// SIMATIC S7-200 project (STEP 7-Micro/WIN), CPU 224 REL 02.01

ORGANIZATION_BLOCK MAIN:OB1
TITLE=PROGRAM COMMENTS
BEGIN
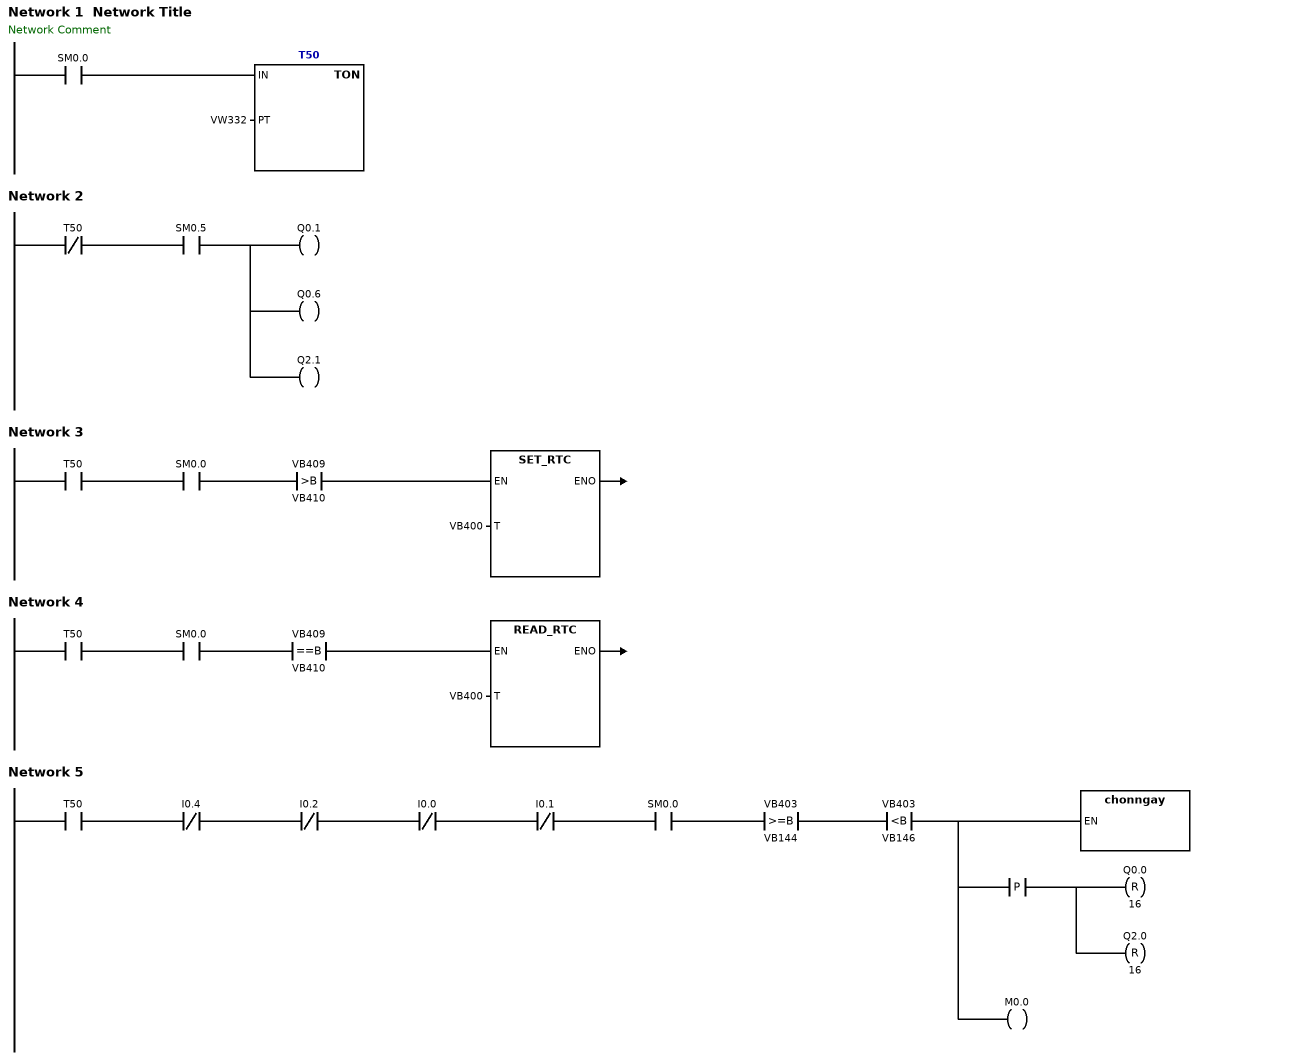
Network 1 // Network Title
// Network Comment
LD     SM0.0
TON    T50, VW332
Network 2
LDN    T50
A      SM0.5
=      Q0.1
=      Q0.6
=      Q2.1
Network 3
LD     T50
A      SM0.0
AB>    VB409, VB410
TODW   VB400
Network 4
LD     T50
A      SM0.0
AB=    VB409, VB410
TODR   VB400
Network 5
LD     T50
AN     I0.4
AN     I0.2
AN     I0.0
AN     I0.1
A      SM0.0
AB>=   VB403, VB144
AB<    VB403, VB146
LPS
CALL   chonngay:SBR11
EU
R      Q0.0, 16
R      Q2.0, 16
LPP
=      M0.0
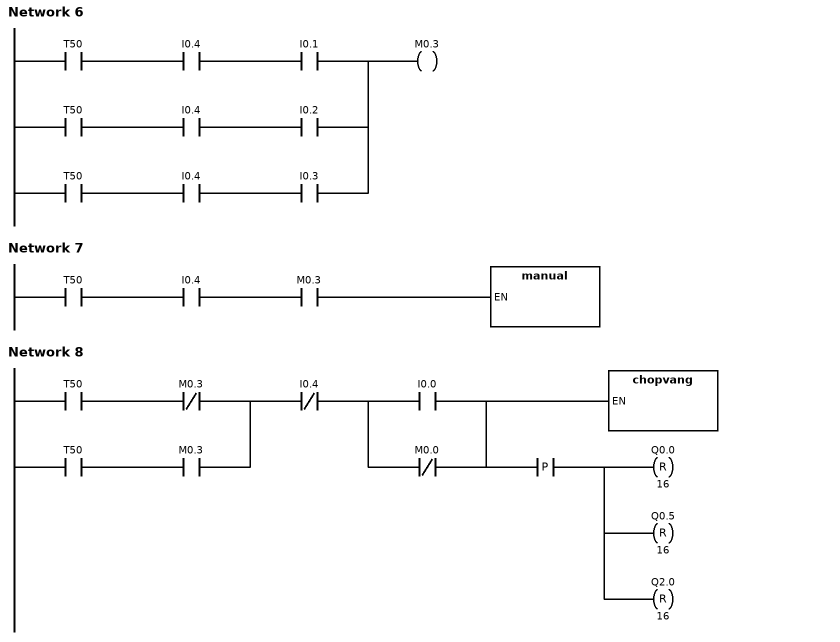
Network 6
LD     T50
A      I0.4
A      I0.1
LD     T50
A      I0.4
A      I0.2
OLD
LD     T50
A      I0.4
A      I0.3
OLD
=      M0.3
Network 7
LD     T50
A      I0.4
A      M0.3
CALL   manual:SBR2
Network 8
LD     T50
AN     M0.3
LD     T50
A      M0.3
OLD
AN     I0.4
LD     I0.0
ON     M0.0
ALD
CALL   chopvang:SBR1
EU
R      Q0.0, 16
R      Q0.5, 16
R      Q2.0, 16
END_ORGANIZATION_BLOCK

SUBROUTINE_BLOCK tudong2phase:SBR0
TITLE=SUBROUTINE COMMENTS
BEGIN
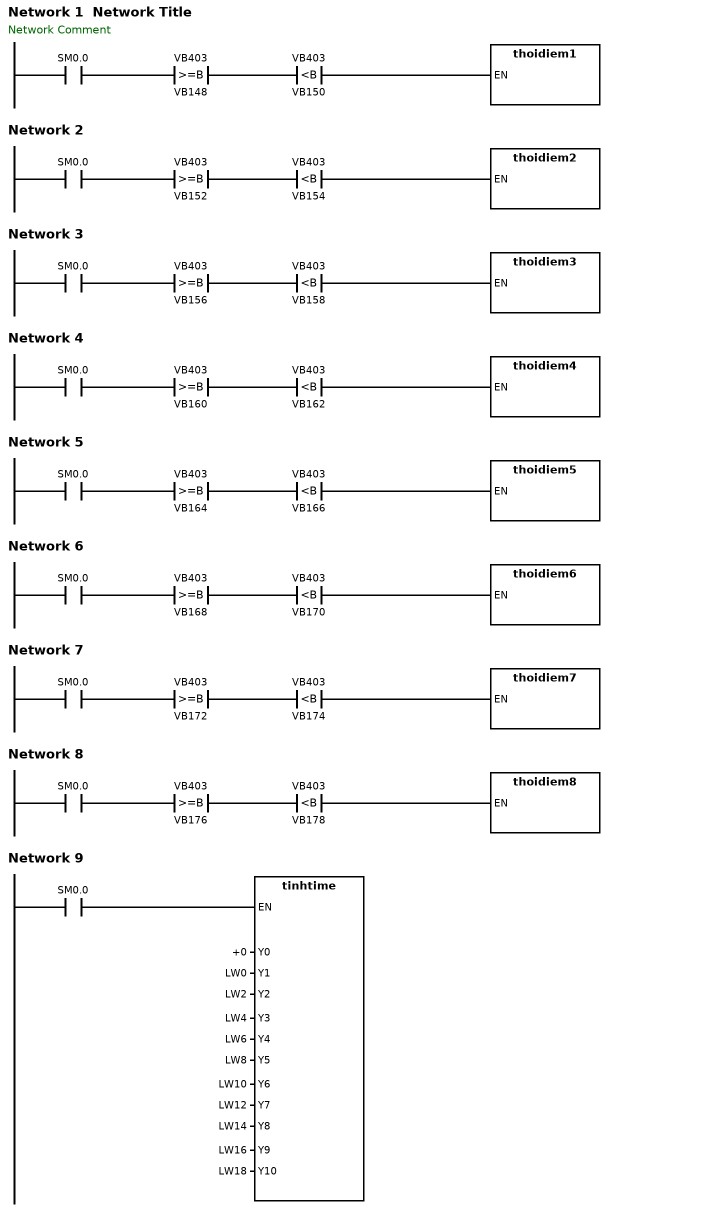
Network 1 // Network Title
// Network Comment
LD     SM0.0
AB>=   VB403, VB148
AB<    VB403, VB150
CALL   thoidiem1:SBR3
Network 2
LD     SM0.0
AB>=   VB403, VB152
AB<    VB403, VB154
CALL   thoidiem2:SBR4
Network 3
LD     SM0.0
AB>=   VB403, VB156
AB<    VB403, VB158
CALL   thoidiem3:SBR5
Network 4
LD     SM0.0
AB>=   VB403, VB160
AB<    VB403, VB162
CALL   thoidiem4:SBR6
Network 5
LD     SM0.0
AB>=   VB403, VB164
AB<    VB403, VB166
CALL   thoidiem5:SBR7
Network 6
LD     SM0.0
AB>=   VB403, VB168
AB<    VB403, VB170
CALL   thoidiem6:SBR8
Network 7
LD     SM0.0
AB>=   VB403, VB172
AB<    VB403, VB174
CALL   thoidiem7:SBR9
Network 8
LD     SM0.0
AB>=   VB403, VB176
AB<    VB403, VB178
CALL   thoidiem8:SBR14
Network 9
LD     SM0.0
CALL   tinhtime:SBR16, +0, LW0, LW2, LW4, LW6, LW8, LW10, LW12, LW14, LW16, LW18
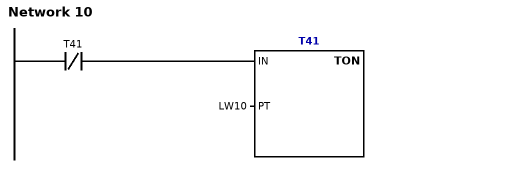
Network 10
LDN    T41
TON    T41, LW10
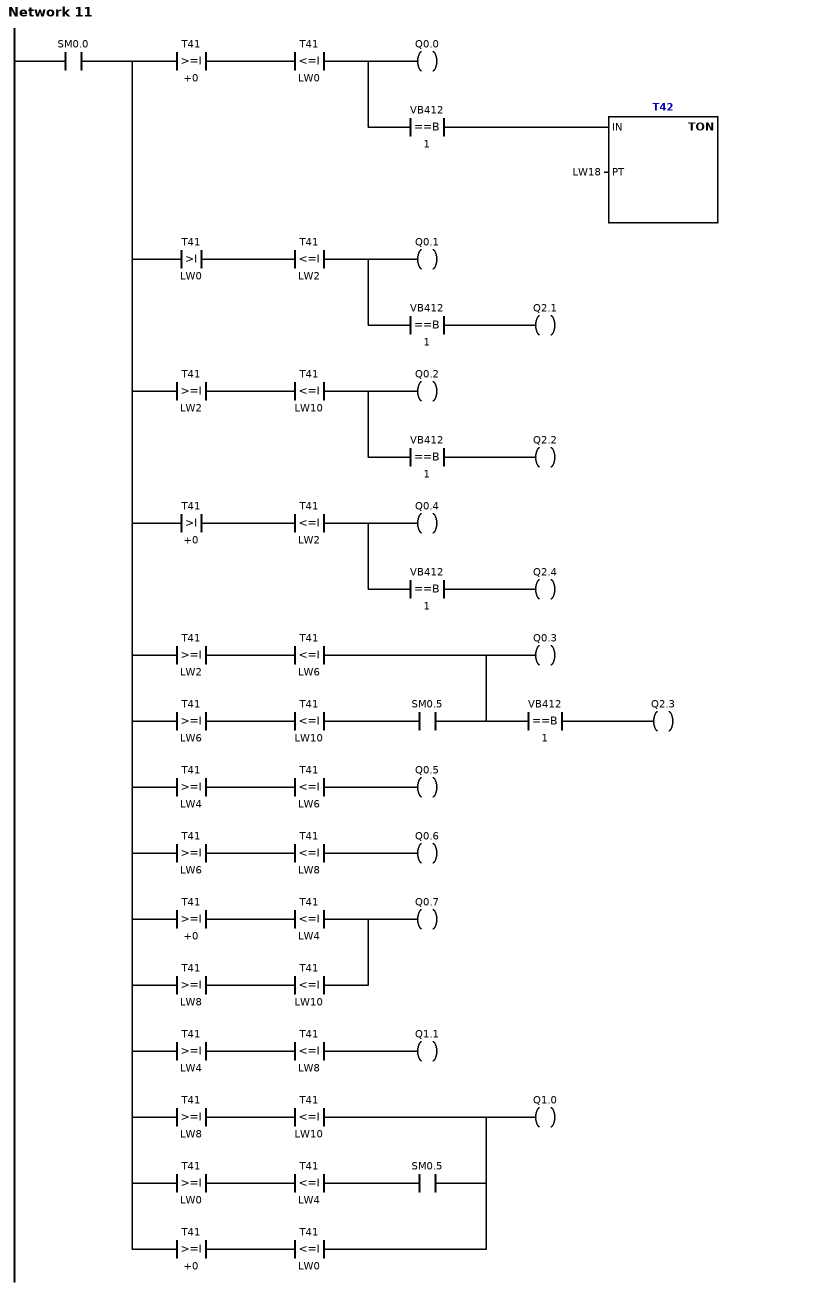
Network 11
LD     SM0.0
LPS
AW>=   T41, +0
AW<=   T41, LW0
=      Q0.0
AB=    VB412, 1
TON    T42, LW18
LRD
AW>    T41, LW0
AW<=   T41, LW2
=      Q0.1
AB=    VB412, 1
=      Q2.1
LRD
AW>=   T41, LW2
AW<=   T41, LW10
=      Q0.2
AB=    VB412, 1
=      Q2.2
LRD
AW>    T41, +0
AW<=   T41, LW2
=      Q0.4
AB=    VB412, 1
=      Q2.4
LRD
LDW>=  T41, LW2
AW<=   T41, LW6
LDW>=  T41, LW6
AW<=   T41, LW10
A      SM0.5
OLD
ALD
=      Q0.3
AB=    VB412, 1
=      Q2.3
LRD
LPS
AW>=   T41, LW4
AW<=   T41, LW6
=      Q0.5
LPP
AW>=   T41, LW6
AW<=   T41, LW8
=      Q0.6
LRD
LDW>=  T41, +0
AW<=   T41, LW4
LDW>=  T41, LW8
AW<=   T41, LW10
OLD
ALD
=      Q0.7
LRD
AW>=   T41, LW4
AW<=   T41, LW8
=      Q1.1
LPP
LDW>=  T41, LW8
AW<=   T41, LW10
LDW>=  T41, LW0
AW<=   T41, LW4
A      SM0.5
OLD
LDW>=  T41, +0
AW<=   T41, LW0
OLD
ALD
=      Q1.0
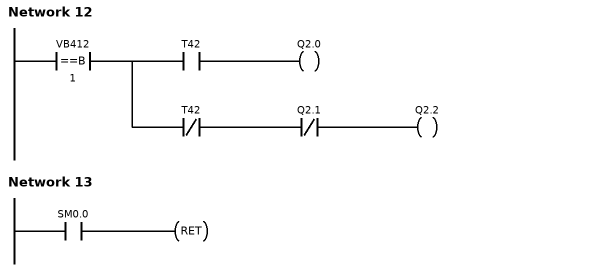
Network 12
LDB=   VB412, 1
LPS
A      T42
=      Q2.0
LPP
AN     T42
AN     Q2.1
=      Q2.2
Network 13
LD     SM0.0
CRET
END_SUBROUTINE_BLOCK

SUBROUTINE_BLOCK chopvang:SBR1
TITLE=
BEGIN
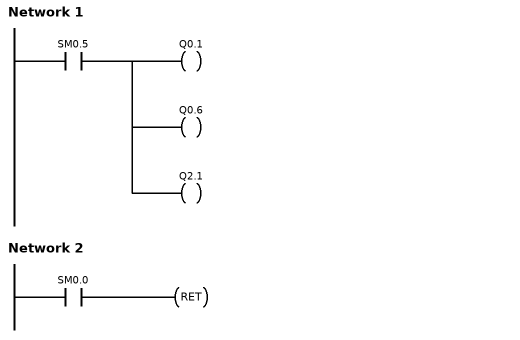
Network 1
LD     SM0.5
=      Q0.1
=      Q0.6
=      Q2.1
Network 2
LD     SM0.0
CRET
END_SUBROUTINE_BLOCK

SUBROUTINE_BLOCK manual:SBR2
TITLE=
BEGIN
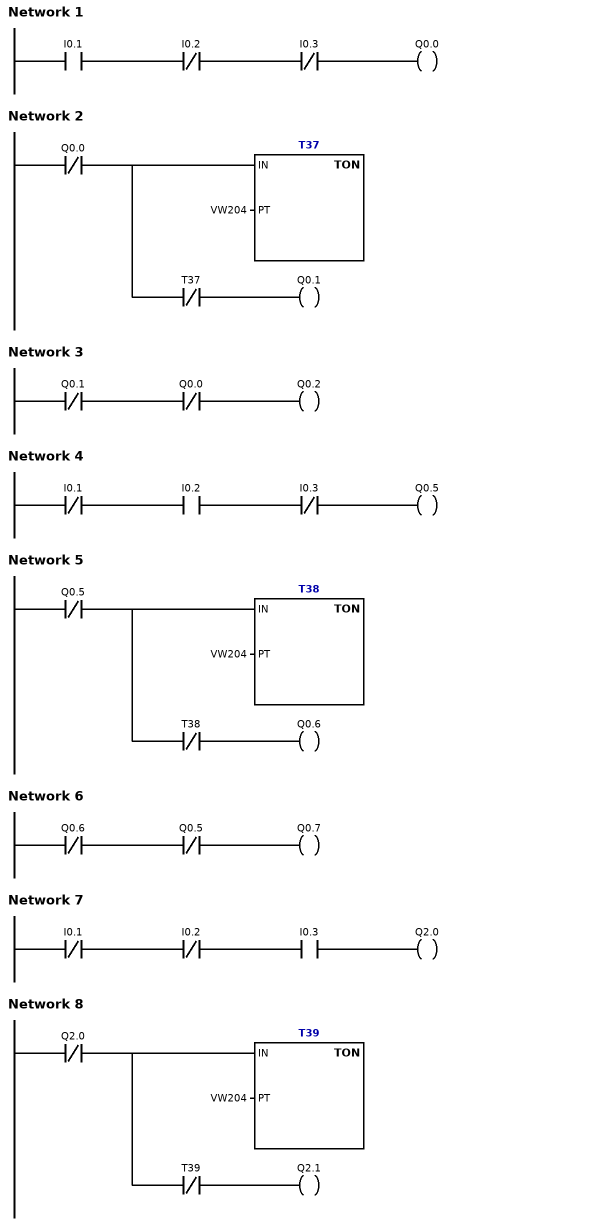
Network 1
LD     I0.1
AN     I0.2
AN     I0.3
=      Q0.0
Network 2
LDN    Q0.0
TON    T37, VW204
AN     T37
=      Q0.1
Network 3
LDN    Q0.1
AN     Q0.0
=      Q0.2
Network 4
LDN    I0.1
A      I0.2
AN     I0.3
=      Q0.5
Network 5
LDN    Q0.5
TON    T38, VW204
AN     T38
=      Q0.6
Network 6
LDN    Q0.6
AN     Q0.5
=      Q0.7
Network 7
LDN    I0.1
AN     I0.2
A      I0.3
=      Q2.0
Network 8
LDN    Q2.0
TON    T39, VW204
AN     T39
=      Q2.1
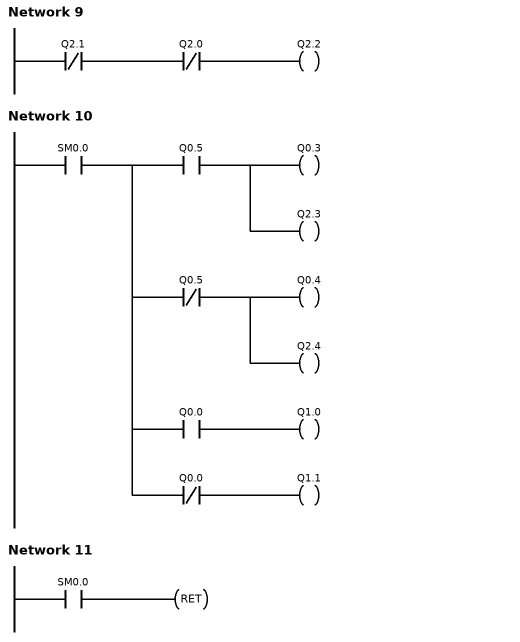
Network 9
LDN    Q2.1
AN     Q2.0
=      Q2.2
Network 10
LD     SM0.0
LPS
A      Q0.5
=      Q0.3
=      Q2.3
LRD
AN     Q0.5
=      Q0.4
=      Q2.4
LPP
LPS
A      Q0.0
=      Q1.0
LPP
AN     Q0.0
=      Q1.1
Network 11
LD     SM0.0
CRET
END_SUBROUTINE_BLOCK

SUBROUTINE_BLOCK thoidiem1:SBR3
TITLE=
BEGIN
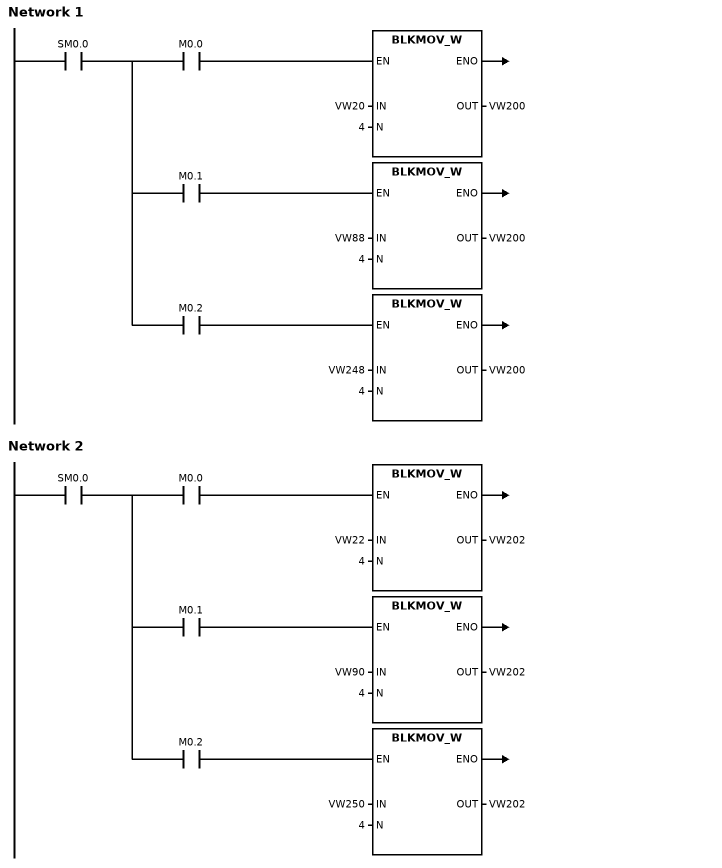
Network 1
LD     SM0.0
LPS
A      M0.0
BMW    VW20, VW200, 4
LRD
A      M0.1
BMW    VW88, VW200, 4
LPP
A      M0.2
BMW    VW248, VW200, 4
Network 2
LD     SM0.0
LPS
A      M0.0
BMW    VW22, VW202, 4
LRD
A      M0.1
BMW    VW90, VW202, 4
LPP
A      M0.2
BMW    VW250, VW202, 4
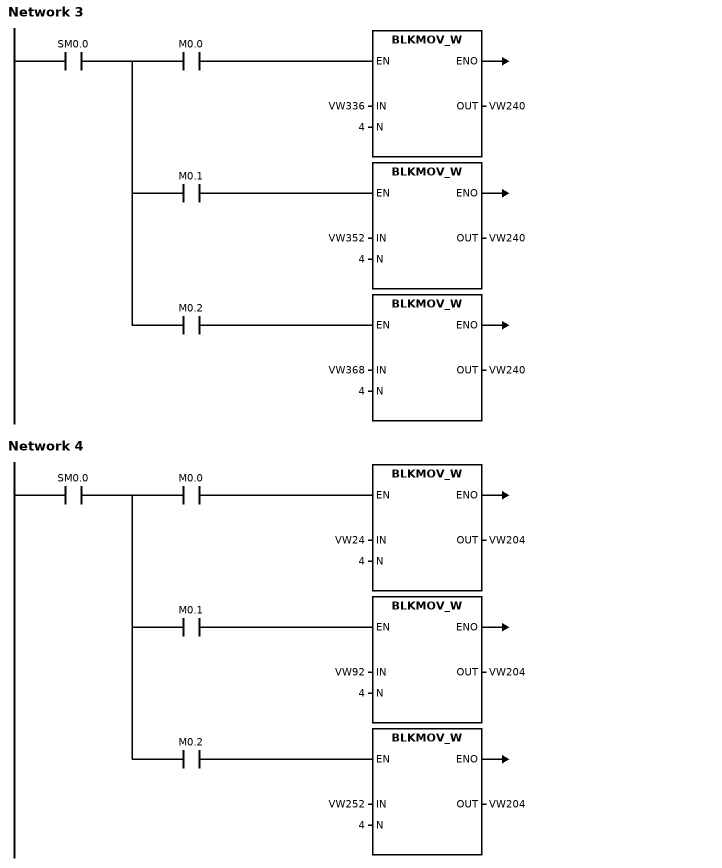
Network 3
LD     SM0.0
LPS
A      M0.0
BMW    VW336, VW240, 4
LRD
A      M0.1
BMW    VW352, VW240, 4
LPP
A      M0.2
BMW    VW368, VW240, 4
Network 4
LD     SM0.0
LPS
A      M0.0
BMW    VW24, VW204, 4
LRD
A      M0.1
BMW    VW92, VW204, 4
LPP
A      M0.2
BMW    VW252, VW204, 4
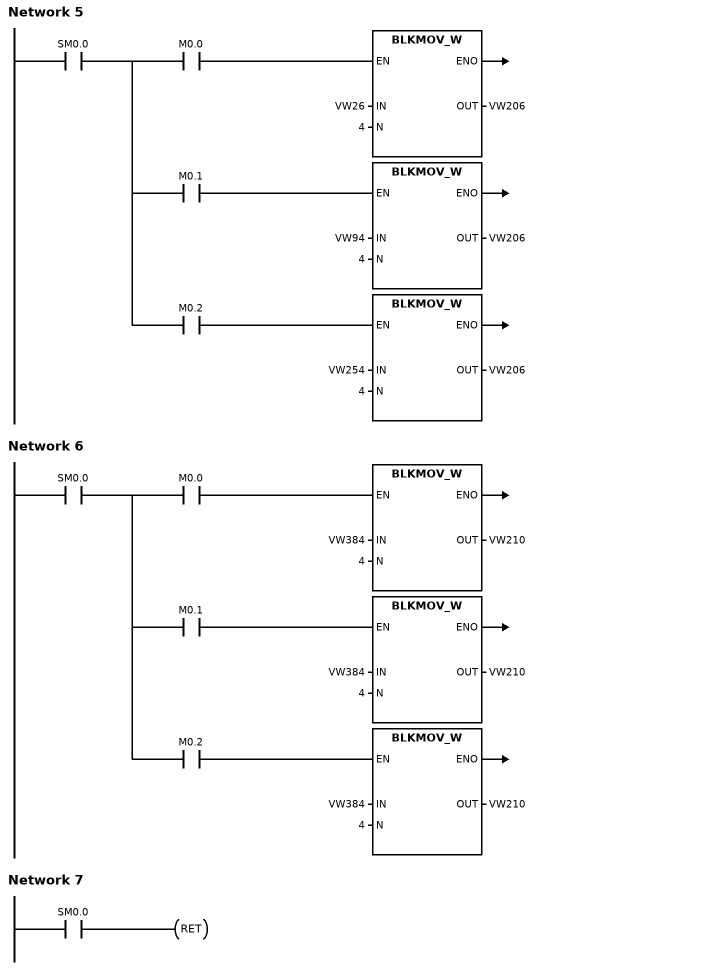
Network 5
LD     SM0.0
LPS
A      M0.0
BMW    VW26, VW206, 4
LRD
A      M0.1
BMW    VW94, VW206, 4
LPP
A      M0.2
BMW    VW254, VW206, 4
Network 6
LD     SM0.0
LPS
A      M0.0
BMW    VW384, VW210, 4
LRD
A      M0.1
BMW    VW384, VW210, 4
LPP
A      M0.2
BMW    VW384, VW210, 4
Network 7
LD     SM0.0
CRET
END_SUBROUTINE_BLOCK

SUBROUTINE_BLOCK thoidiem2:SBR4
TITLE=
BEGIN
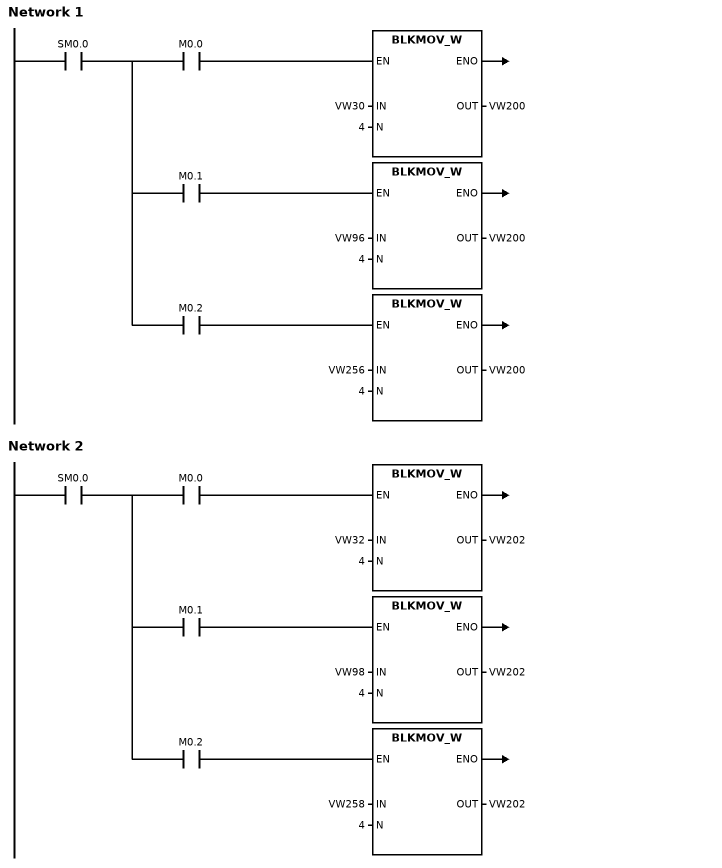
Network 1
LD     SM0.0
LPS
A      M0.0
BMW    VW30, VW200, 4
LRD
A      M0.1
BMW    VW96, VW200, 4
LPP
A      M0.2
BMW    VW256, VW200, 4
Network 2
LD     SM0.0
LPS
A      M0.0
BMW    VW32, VW202, 4
LRD
A      M0.1
BMW    VW98, VW202, 4
LPP
A      M0.2
BMW    VW258, VW202, 4
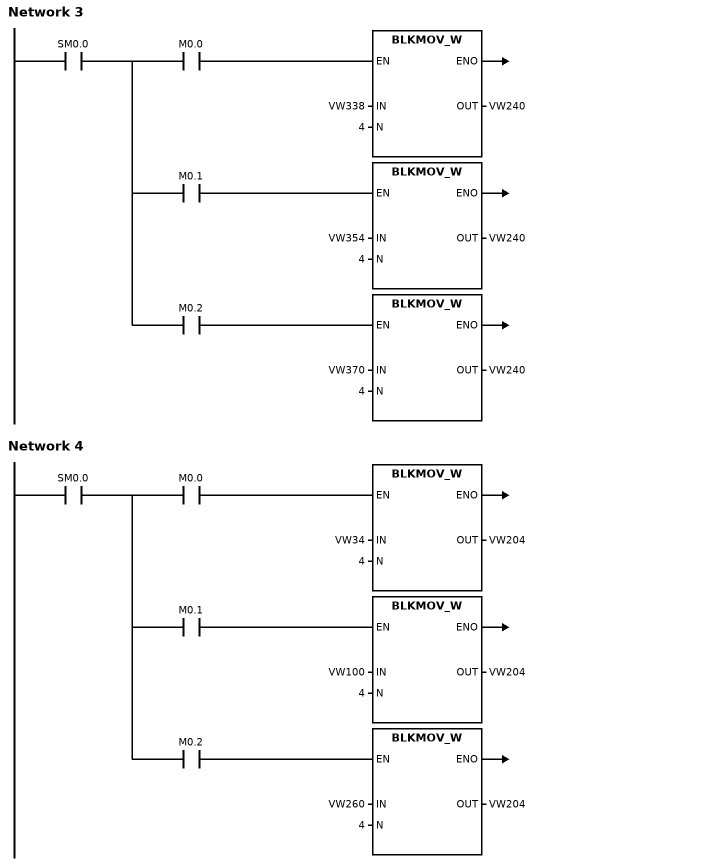
Network 3
LD     SM0.0
LPS
A      M0.0
BMW    VW338, VW240, 4
LRD
A      M0.1
BMW    VW354, VW240, 4
LPP
A      M0.2
BMW    VW370, VW240, 4
Network 4
LD     SM0.0
LPS
A      M0.0
BMW    VW34, VW204, 4
LRD
A      M0.1
BMW    VW100, VW204, 4
LPP
A      M0.2
BMW    VW260, VW204, 4
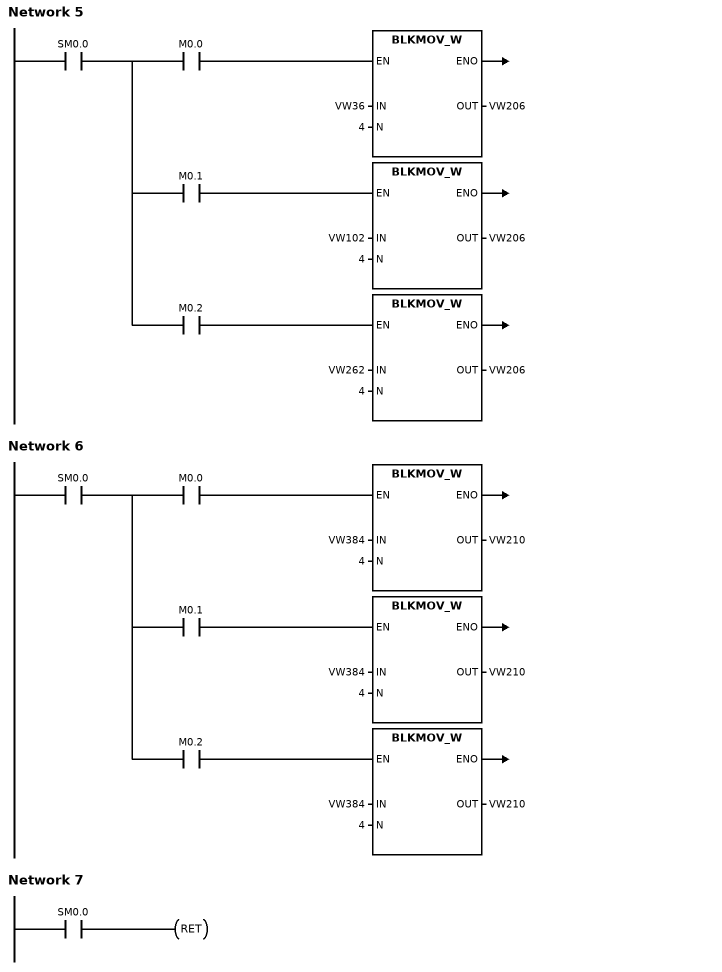
Network 5
LD     SM0.0
LPS
A      M0.0
BMW    VW36, VW206, 4
LRD
A      M0.1
BMW    VW102, VW206, 4
LPP
A      M0.2
BMW    VW262, VW206, 4
Network 6
LD     SM0.0
LPS
A      M0.0
BMW    VW384, VW210, 4
LRD
A      M0.1
BMW    VW384, VW210, 4
LPP
A      M0.2
BMW    VW384, VW210, 4
Network 7
LD     SM0.0
CRET
END_SUBROUTINE_BLOCK

SUBROUTINE_BLOCK thoidiem3:SBR5
TITLE=
BEGIN
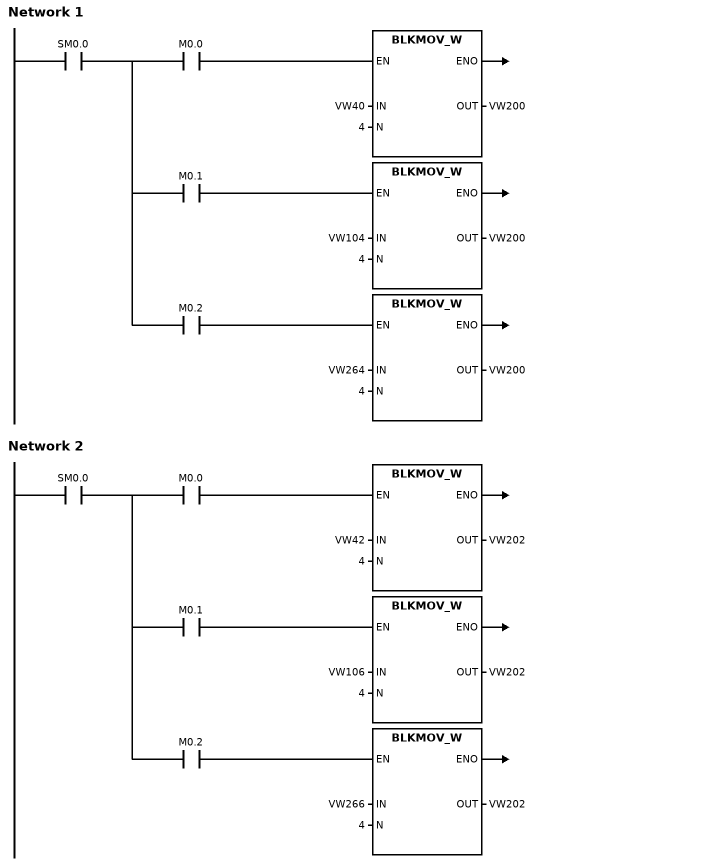
Network 1
LD     SM0.0
LPS
A      M0.0
BMW    VW40, VW200, 4
LRD
A      M0.1
BMW    VW104, VW200, 4
LPP
A      M0.2
BMW    VW264, VW200, 4
Network 2
LD     SM0.0
LPS
A      M0.0
BMW    VW42, VW202, 4
LRD
A      M0.1
BMW    VW106, VW202, 4
LPP
A      M0.2
BMW    VW266, VW202, 4
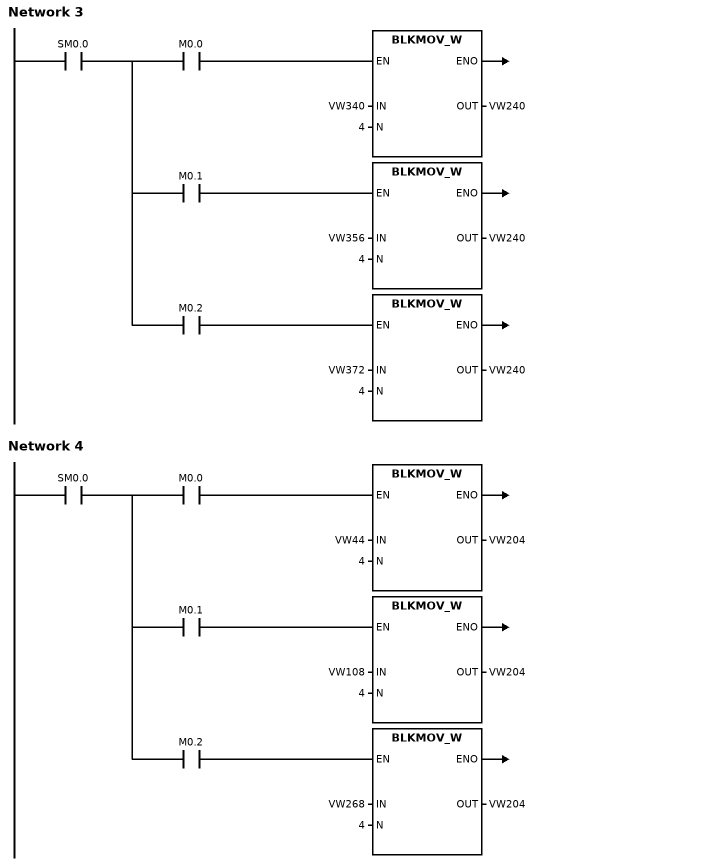
Network 3
LD     SM0.0
LPS
A      M0.0
BMW    VW340, VW240, 4
LRD
A      M0.1
BMW    VW356, VW240, 4
LPP
A      M0.2
BMW    VW372, VW240, 4
Network 4
LD     SM0.0
LPS
A      M0.0
BMW    VW44, VW204, 4
LRD
A      M0.1
BMW    VW108, VW204, 4
LPP
A      M0.2
BMW    VW268, VW204, 4
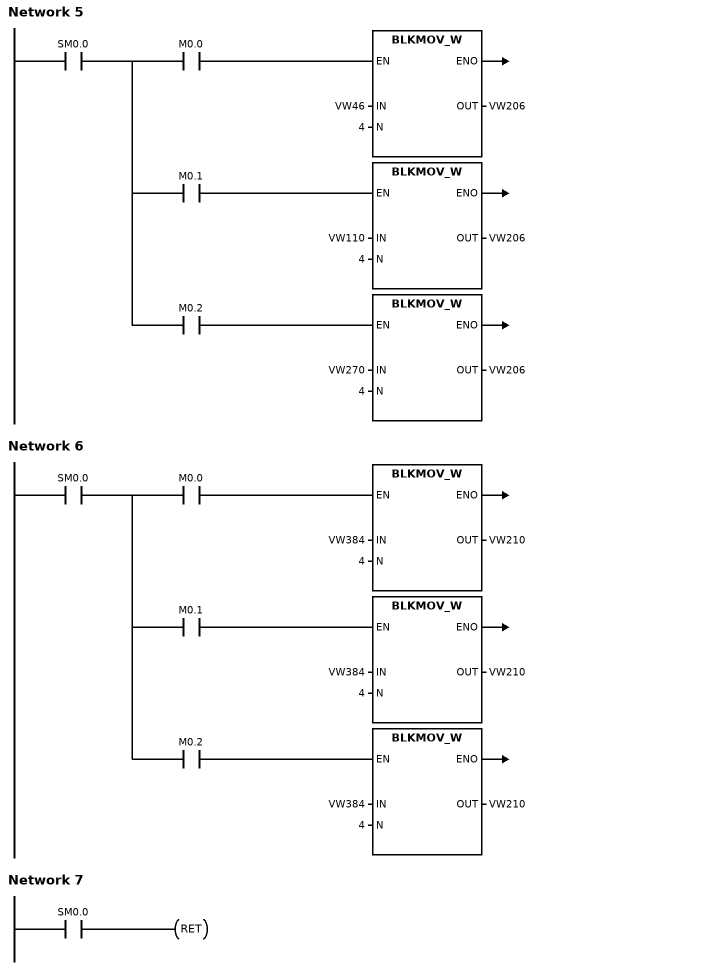
Network 5
LD     SM0.0
LPS
A      M0.0
BMW    VW46, VW206, 4
LRD
A      M0.1
BMW    VW110, VW206, 4
LPP
A      M0.2
BMW    VW270, VW206, 4
Network 6
LD     SM0.0
LPS
A      M0.0
BMW    VW384, VW210, 4
LRD
A      M0.1
BMW    VW384, VW210, 4
LPP
A      M0.2
BMW    VW384, VW210, 4
Network 7
LD     SM0.0
CRET
END_SUBROUTINE_BLOCK

SUBROUTINE_BLOCK thoidiem4:SBR6
TITLE=
BEGIN
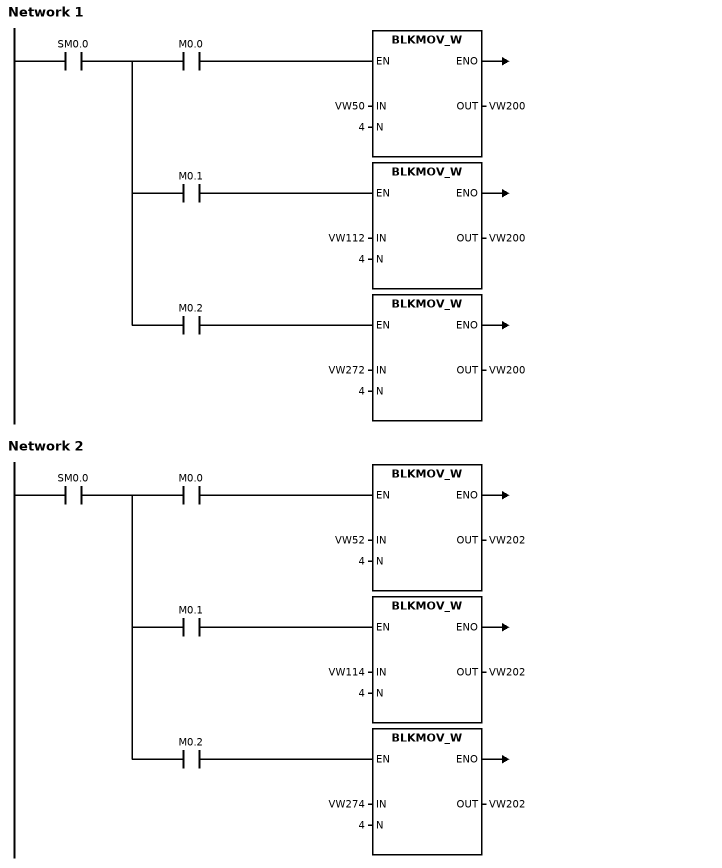
Network 1
LD     SM0.0
LPS
A      M0.0
BMW    VW50, VW200, 4
LRD
A      M0.1
BMW    VW112, VW200, 4
LPP
A      M0.2
BMW    VW272, VW200, 4
Network 2
LD     SM0.0
LPS
A      M0.0
BMW    VW52, VW202, 4
LRD
A      M0.1
BMW    VW114, VW202, 4
LPP
A      M0.2
BMW    VW274, VW202, 4
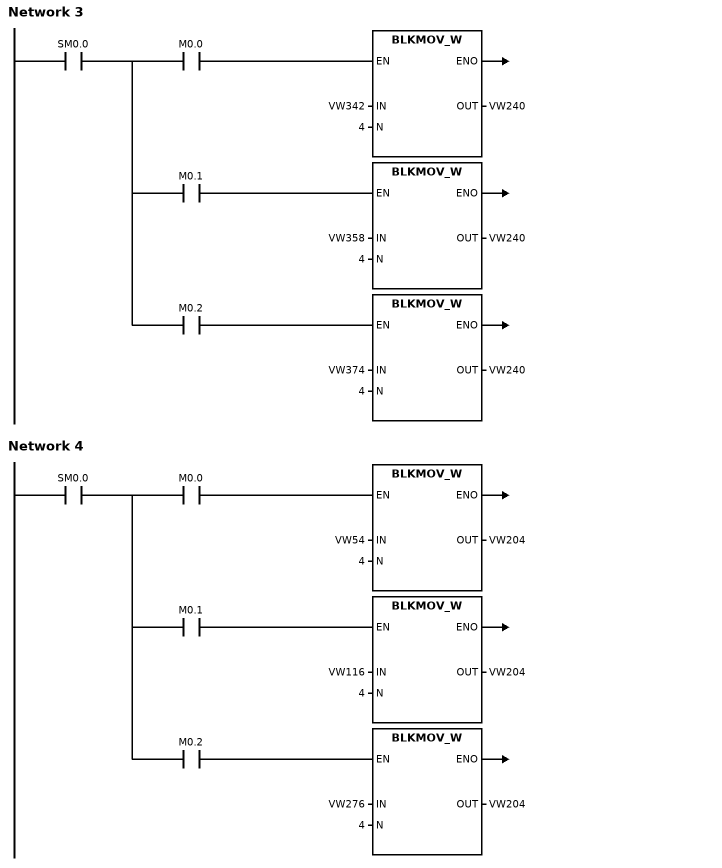
Network 3
LD     SM0.0
LPS
A      M0.0
BMW    VW342, VW240, 4
LRD
A      M0.1
BMW    VW358, VW240, 4
LPP
A      M0.2
BMW    VW374, VW240, 4
Network 4
LD     SM0.0
LPS
A      M0.0
BMW    VW54, VW204, 4
LRD
A      M0.1
BMW    VW116, VW204, 4
LPP
A      M0.2
BMW    VW276, VW204, 4
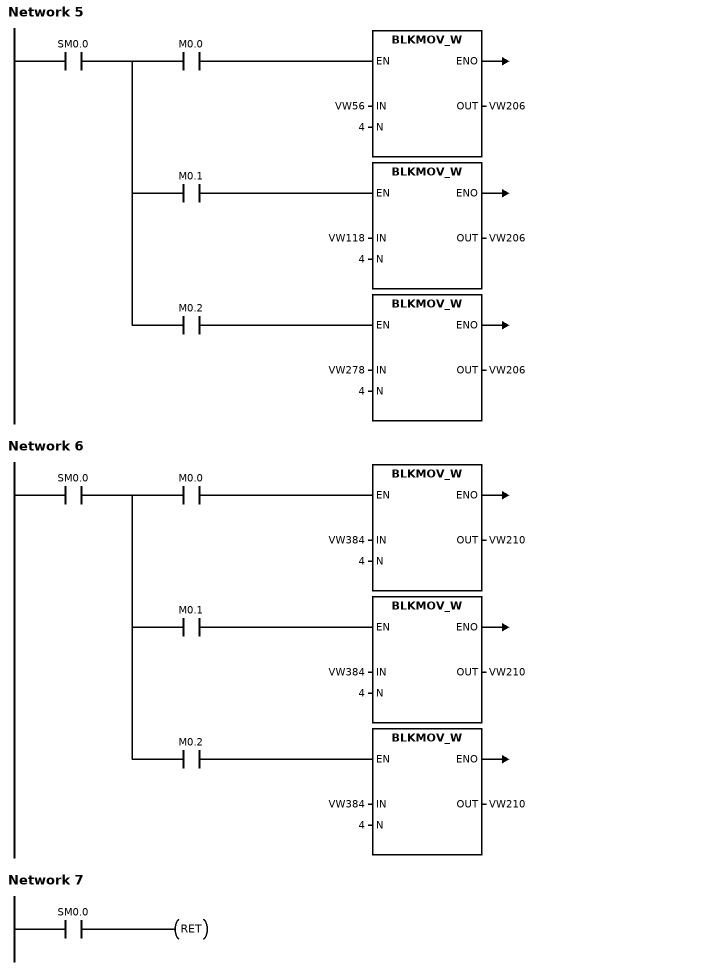
Network 5
LD     SM0.0
LPS
A      M0.0
BMW    VW56, VW206, 4
LRD
A      M0.1
BMW    VW118, VW206, 4
LPP
A      M0.2
BMW    VW278, VW206, 4
Network 6
LD     SM0.0
LPS
A      M0.0
BMW    VW384, VW210, 4
LRD
A      M0.1
BMW    VW384, VW210, 4
LPP
A      M0.2
BMW    VW384, VW210, 4
Network 7
LD     SM0.0
CRET
END_SUBROUTINE_BLOCK

SUBROUTINE_BLOCK thoidiem5:SBR7
TITLE=
BEGIN
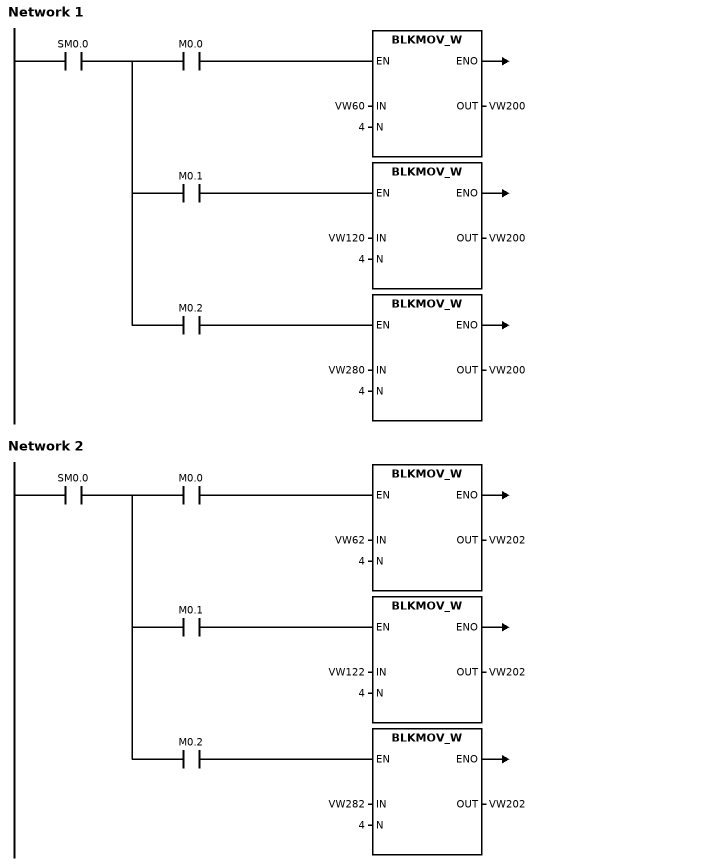
Network 1
LD     SM0.0
LPS
A      M0.0
BMW    VW60, VW200, 4
LRD
A      M0.1
BMW    VW120, VW200, 4
LPP
A      M0.2
BMW    VW280, VW200, 4
Network 2
LD     SM0.0
LPS
A      M0.0
BMW    VW62, VW202, 4
LRD
A      M0.1
BMW    VW122, VW202, 4
LPP
A      M0.2
BMW    VW282, VW202, 4
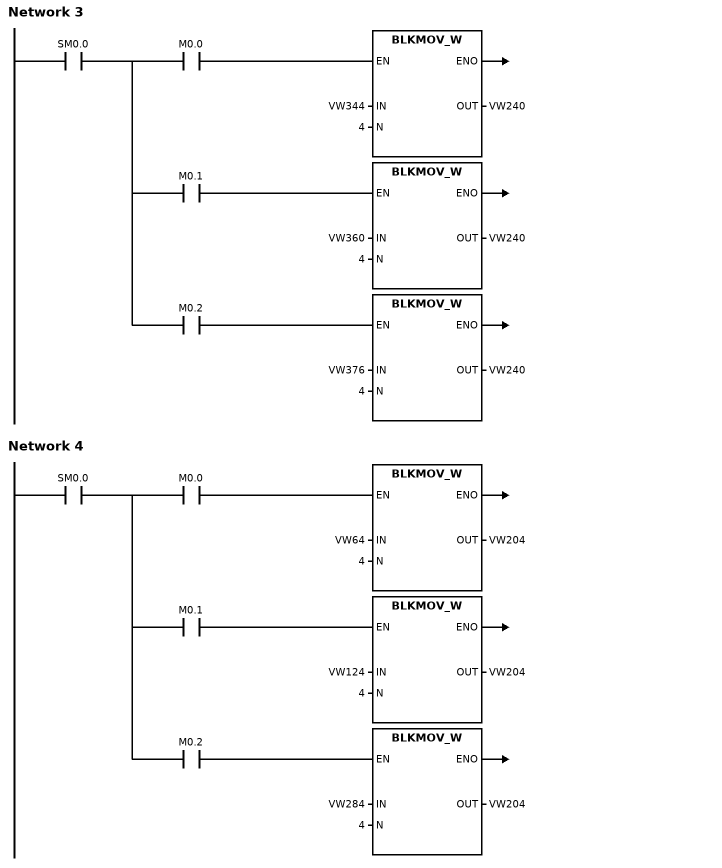
Network 3
LD     SM0.0
LPS
A      M0.0
BMW    VW344, VW240, 4
LRD
A      M0.1
BMW    VW360, VW240, 4
LPP
A      M0.2
BMW    VW376, VW240, 4
Network 4
LD     SM0.0
LPS
A      M0.0
BMW    VW64, VW204, 4
LRD
A      M0.1
BMW    VW124, VW204, 4
LPP
A      M0.2
BMW    VW284, VW204, 4
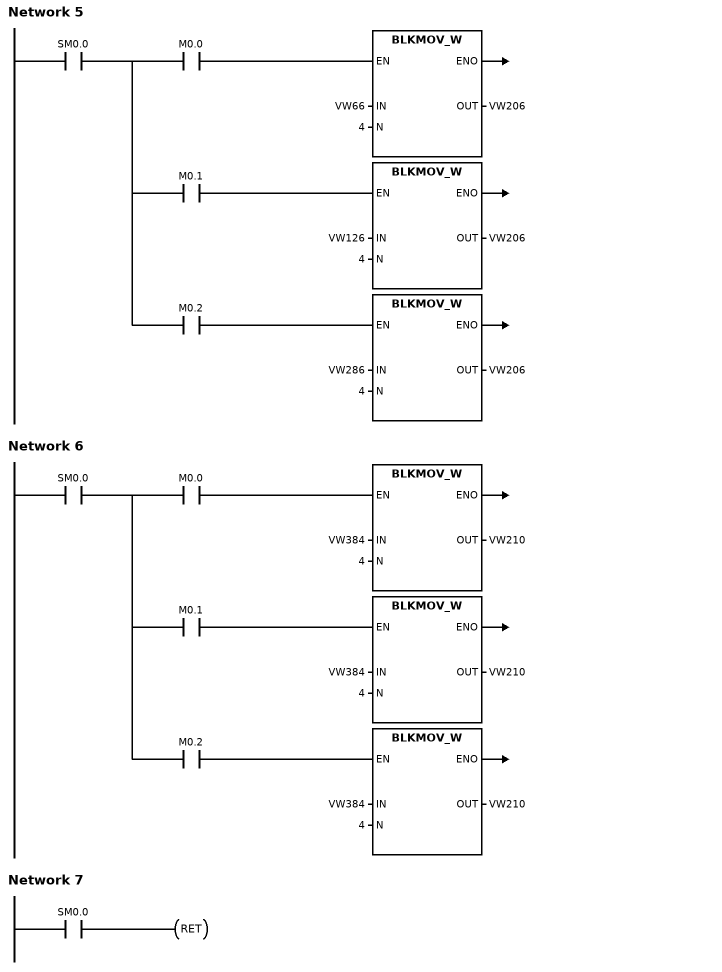
Network 5
LD     SM0.0
LPS
A      M0.0
BMW    VW66, VW206, 4
LRD
A      M0.1
BMW    VW126, VW206, 4
LPP
A      M0.2
BMW    VW286, VW206, 4
Network 6
LD     SM0.0
LPS
A      M0.0
BMW    VW384, VW210, 4
LRD
A      M0.1
BMW    VW384, VW210, 4
LPP
A      M0.2
BMW    VW384, VW210, 4
Network 7
LD     SM0.0
CRET
END_SUBROUTINE_BLOCK

SUBROUTINE_BLOCK thoidiem6:SBR8
TITLE=
BEGIN
